PROGRAM PMPS_Arbiter
VAR
	
	
	fbMachine	:	FB_MachineSimulator;
	
	fbMPSInterface	:	FB_BeamClassOutputs;
END_VAR


//Execute arbiter
fbArbiter();

fbMPSInterface();

//Machine simulator
fbMachine(
	i_stAssertedParams := fbArbiter.q_stBeamParams,
	q_stMachineParams => PMPS_GVL_BeamParams.stCurrentBeamParameters
	);

END_PROGRAM

(* stored: Version 1.1.0.1, ProductVersion 3.1.4022.12
   POU PMPS_Arbiter: Id {91ae890b-11cc-4d41-83ec-edc5b802c784}, SpecialFunc None *)
